(* PLC project tc_project_app, Beckhoff Automation GmbH TwinCAT PLC Control 3.5.13.21 *)
(* stored: creationDateTime 2023-08-04T14:20:43.0098278, modificationDateTime 2023-08-04T14:20:43.0127944 *)

PROGRAM Axis_Template
VAR
//Outputs: Power for Limit switches, Home Sensors, etc.
    //bPowerSwitchesAxis1 AT %Q*: BOOL:= TRUE;

//Hardware interlocks
    //bInterlockFwdOK AT %I*: BOOL;
END_VAR

            //Initial parameters of an Axis
(*IF _TaskInfo[fbGetCurTaskIndex.index].FirstCycle THEN
    //Axis description for EPICS PV
    GVL.astAxes[1].stDescription.sAxisName := 'MotorApplication1';
    GVL.astAxes[1].stDescription.eUnit := E_AxisEngUnit.eMeter;
    GVL.astAxes[1].stDescription.nPrefix := -3;

    //Initial default values:
    GVL.astAxes[1].stConfig.eHomeSeq := 0;
    GVL.astAxes[1].stConfig.fHomePosition := 0.0;
    GVL.astAxes[1].stConfig.fHomeFinishDistance := 0.0;
    GVL.astAxes[1].stConfig.eRestorePosition := E_RestorePosition.eRestoreWithoutHome;
END_IF*)

//Define ACTIONS() or write exclusive code for an specific axis.
(*Eg. Stop when temperature reaches certain values, reduce speed if  a signal is activated, etc.
Eg. GVL.astAxes[x].stControl.bInterlockFwd := NOT bInterlockFwdOK;*)

          
END_PROGRAM
